DATA_BLOCK "SettingsDB"
{ S7_Optimized_Access := 'FALSE'; DB_Accessible_From_OPC_UA := 'TRUE' }
VERSION : '1.0'
READ_ONLY
VAR RETAIN
    CONFIG : "Config_001";
    MAINTENANCE_MODE : BOOL;
    MAINTENANCE_TIMEOUT : TIME;
END_VAR
BEGIN
    MAINTENANCE_MODE := FALSE;
    MAINTENANCE_TIMEOUT := T#1h;
    CONFIG.DINT_VAL := 42;
    CONFIG.INT_ARRAY[0] := 1;
    CONFIG.INT_ARRAY[1] := 2;
    CONFIG.INT_ARRAY[2] := 3;
    CONFIG.REAL_ARRAY[0] := 1.1;
    CONFIG.REAL_ARRAY[1] := 2.2;
    CONFIG.REAL_ARRAY[2] := 3.3;
END_DATA_BLOCK